// TIA Portal V20 export
FUNCTION "CollectAlarms" : Void   // FC85, LAD
TITLE = Alarm Collector Unit
// Collects alarms from the respective level and categorises the alarms into the different alarm classes.
// stored: Namespace Unit1.Em7, SetENOAutomatically false
   VAR_INPUT
      resetAlarms : Bool;
      disableAlarms : Bool;
   END_VAR
   VAR_OUTPUT
      commandsToUnit : "LUC_typeStateCommands";   // Feedback to the unit
   END_VAR
   VAR CONSTANT
      DelayTime : Time := T#100ms;
      NoDelayTime : Time;
      TRUE : Bool := TRUE;
      FALSE : Bool := FALSE;
   END_VAR
   VAR_TEMP   // added for the SCL form of the ladder/FBD networks
      _w1 : Bool;
   END_VAR
BEGIN

REGION Network 1: Reset Alarms
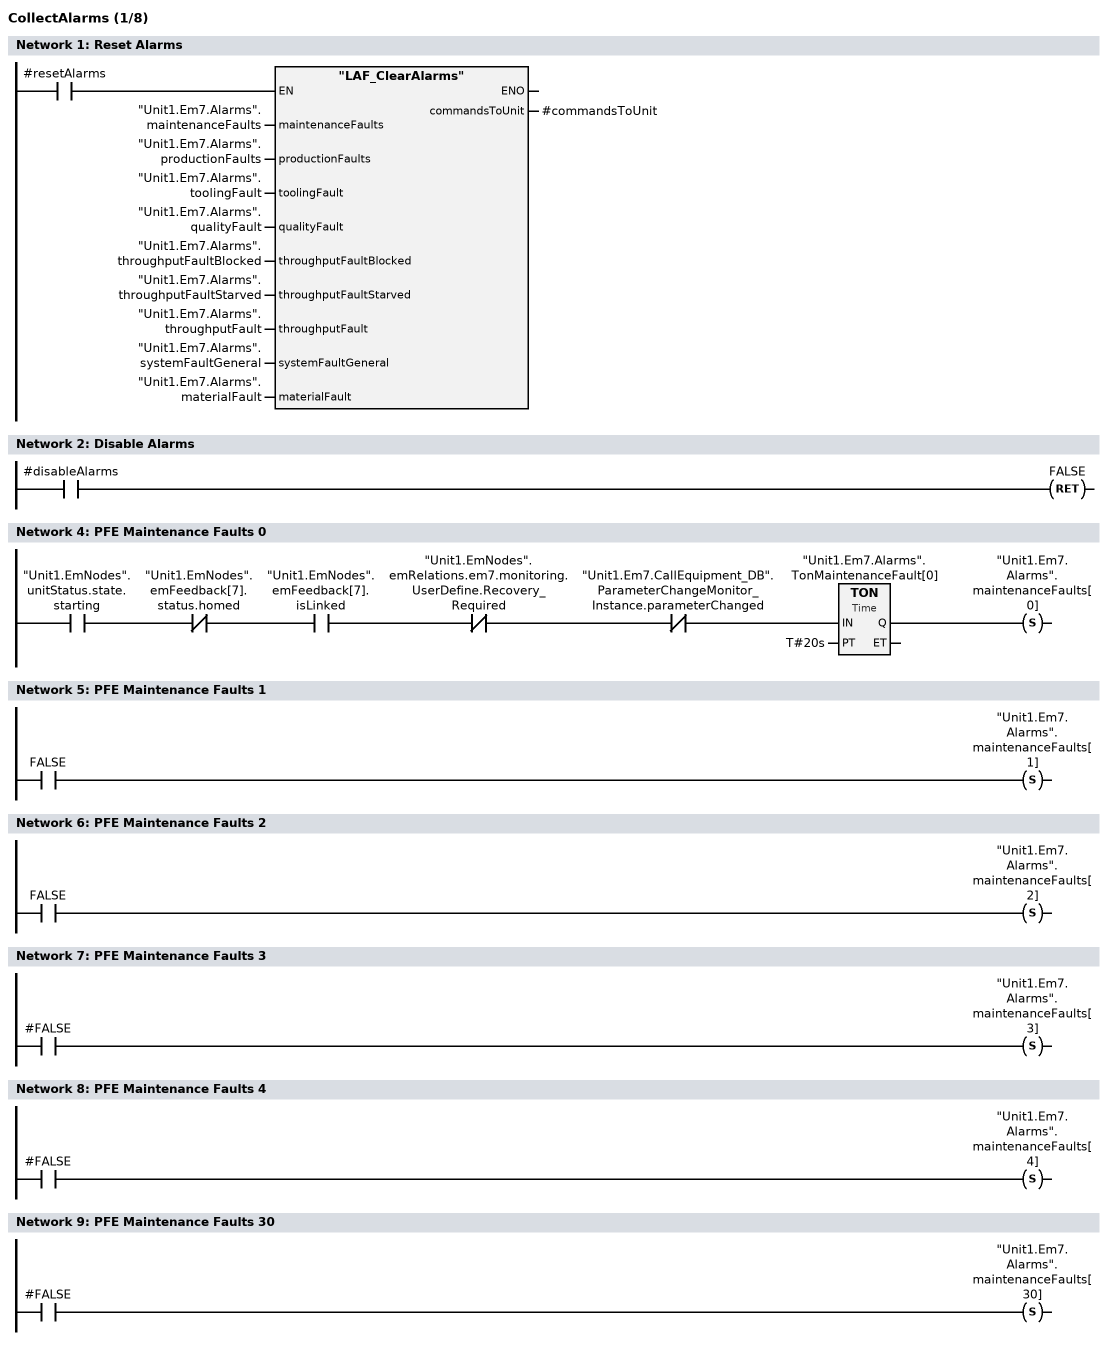
   RUNG wire#powerrail
      Contact( #resetAlarms )
      "LAF_ClearAlarms"(maintenanceFaults := "Unit1.Em7.Alarms".maintenanceFaults, productionFaults := "Unit1.Em7.Alarms".productionFaults, toolingFault := "Unit1.Em7.Alarms".toolingFault, qualityFault := "Unit1.Em7.Alarms".qualityFault, throughputFaultBlocked := "Unit1.Em7.Alarms".throughputFaultBlocked, throughputFaultStarved := "Unit1.Em7.Alarms".throughputFaultStarved, throughputFault := "Unit1.Em7.Alarms".throughputFault, systemFaultGeneral := "Unit1.Em7.Alarms".systemFaultGeneral, materialFault := "Unit1.Em7.Alarms".materialFault, commandsToUnit => #commandsToUnit)
   END_RUNG
   // the same network as SCL:
   IF #resetAlarms THEN
       "LAF_ClearAlarms"(maintenanceFaults := "Unit1.Em7.Alarms".maintenanceFaults,
                         productionFaults := "Unit1.Em7.Alarms".productionFaults,
                         toolingFault := "Unit1.Em7.Alarms".toolingFault,
                         qualityFault := "Unit1.Em7.Alarms".qualityFault,
                         throughputFaultBlocked := "Unit1.Em7.Alarms".throughputFaultBlocked,
                         throughputFaultStarved := "Unit1.Em7.Alarms".throughputFaultStarved,
                         throughputFault := "Unit1.Em7.Alarms".throughputFault,
                         systemFaultGeneral := "Unit1.Em7.Alarms".systemFaultGeneral,
                         materialFault := "Unit1.Em7.Alarms".materialFault,
                         commandsToUnit => #commandsToUnit);
   END_IF;
END_REGION

REGION Network 2: Disable Alarms
   RUNG wire#powerrail
      Contact( #disableAlarms )
      ReturnCoil( FALSE )
   END_RUNG
   // the same network as SCL:
   IF #disableAlarms THEN
       ENO := FALSE;
       RETURN;
   END_IF;
END_REGION

REGION Network 3: *************** Fault ************************
END_REGION

REGION Network 4: PFE Maintenance Faults 0
   RUNG wire#powerrail
      Contact( "Unit1.EmNodes".unitStatus.state.starting )
      I_Contact( "Unit1.EmNodes".emFeedback[7].status.homed )
      Contact( "Unit1.EmNodes".emFeedback[7].isLinked )
      I_Contact( "Unit1.EmNodes".emRelations.em7.monitoring.UserDefine.Recovery_Required )
      I_Contact( "Unit1.Em7.CallEquipment_DB".ParameterChangeMonitor_Instance.parameterChanged )
      { S7_Templates := "time_type := Time" } "Unit1.Em7.Alarms".TonMaintenanceFault[0].TON(pt := T#20s, et =>)
      S_Coil( "Unit1.Em7.Alarms".maintenanceFaults[0] )
   END_RUNG
   // the same network as SCL:
   "Unit1.Em7.Alarms".TonMaintenanceFault[0].TON(IN := "Unit1.EmNodes".unitStatus.state.starting AND NOT "Unit1.EmNodes".emFeedback[7].status.homed AND "Unit1.EmNodes".emFeedback[7].isLinked AND NOT "Unit1.EmNodes".emRelations.em7.monitoring.UserDefine.Recovery_Required AND NOT "Unit1.Em7.CallEquipment_DB".ParameterChangeMonitor_Instance.parameterChanged,
                           PT := T#20s);
   IF "Unit1.Em7.Alarms".TonMaintenanceFault[0].Q THEN
       "Unit1.Em7.Alarms".maintenanceFaults[0] := TRUE;
   END_IF;
END_REGION

REGION Network 5: PFE Maintenance Faults 1
   RUNG wire#powerrail
      Contact( FALSE )
      S_Coil( "Unit1.Em7.Alarms".maintenanceFaults[1] )
   END_RUNG
   // the same network as SCL:
   IF FALSE THEN "Unit1.Em7.Alarms".maintenanceFaults[1] := TRUE; END_IF;
END_REGION

REGION Network 6: PFE Maintenance Faults 2
   RUNG wire#powerrail
      Contact( FALSE )
      S_Coil( "Unit1.Em7.Alarms".maintenanceFaults[2] )
   END_RUNG
   // the same network as SCL:
   IF FALSE THEN "Unit1.Em7.Alarms".maintenanceFaults[2] := TRUE; END_IF;
END_REGION

REGION Network 7: PFE Maintenance Faults 3
   RUNG wire#powerrail
      Contact( #FALSE )
      S_Coil( "Unit1.Em7.Alarms".maintenanceFaults[3] )
   END_RUNG
   // the same network as SCL:
   IF #FALSE THEN "Unit1.Em7.Alarms".maintenanceFaults[3] := TRUE; END_IF;
END_REGION

REGION Network 8: PFE Maintenance Faults 4
   RUNG wire#powerrail
      Contact( #FALSE )
      S_Coil( "Unit1.Em7.Alarms".maintenanceFaults[4] )
   END_RUNG
   // the same network as SCL:
   IF #FALSE THEN "Unit1.Em7.Alarms".maintenanceFaults[4] := TRUE; END_IF;
END_REGION

REGION Network 9: PFE Maintenance Faults 30
   RUNG wire#powerrail
      Contact( #FALSE )
      S_Coil( "Unit1.Em7.Alarms".maintenanceFaults[30] )
   END_RUNG
   // the same network as SCL:
   IF #FALSE THEN "Unit1.Em7.Alarms".maintenanceFaults[30] := TRUE; END_IF;
END_REGION

REGION Network 10: PFE Maintenance Faults 31
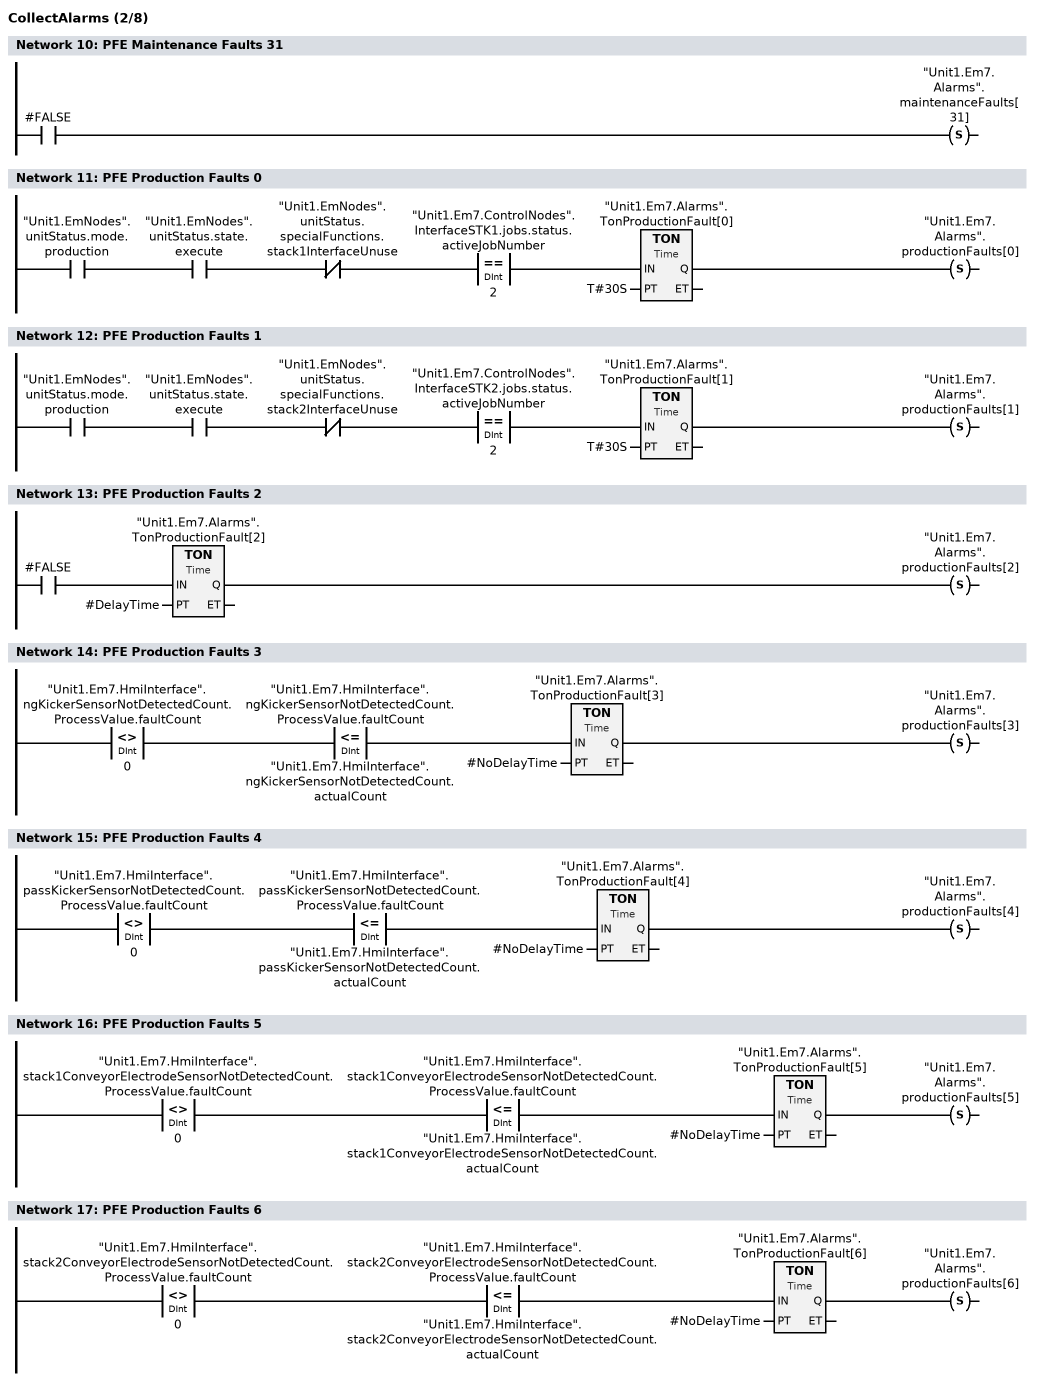
   RUNG wire#powerrail
      Contact( #FALSE )
      S_Coil( "Unit1.Em7.Alarms".maintenanceFaults[31] )
   END_RUNG
   // the same network as SCL:
   IF #FALSE THEN "Unit1.Em7.Alarms".maintenanceFaults[31] := TRUE; END_IF;
END_REGION

REGION Network 11: PFE Production Faults 0
   RUNG wire#powerrail
      Contact( "Unit1.EmNodes".unitStatus.mode.production )
      Contact( "Unit1.EmNodes".unitStatus.state.execute )
      I_Contact( "Unit1.EmNodes".unitStatus.specialFunctions.stack1InterfaceUnuse )
      { S7_Templates := "SrcType := DInt" } EQ_Contact(in1 := "Unit1.Em7.ControlNodes".InterfaceSTK1.jobs.status.activeJobNumber, in2 := 2)
      { S7_Templates := "time_type := Time" } "Unit1.Em7.Alarms".TonProductionFault[0].TON(pt := T#30S, et =>)
      S_Coil( "Unit1.Em7.Alarms".productionFaults[0] )
   END_RUNG
   // the same network as SCL:
   "Unit1.Em7.Alarms".TonProductionFault[0].TON(IN := "Unit1.EmNodes".unitStatus.mode.production AND "Unit1.EmNodes".unitStatus.state.execute AND NOT "Unit1.EmNodes".unitStatus.specialFunctions.stack1InterfaceUnuse AND ("Unit1.Em7.ControlNodes".InterfaceSTK1.jobs.status.activeJobNumber = 2),
                           PT := T#30S);
   IF "Unit1.Em7.Alarms".TonProductionFault[0].Q THEN "Unit1.Em7.Alarms".productionFaults[0] := TRUE; END_IF;
END_REGION

REGION Network 12: PFE Production Faults 1
   RUNG wire#powerrail
      Contact( "Unit1.EmNodes".unitStatus.mode.production )
      Contact( "Unit1.EmNodes".unitStatus.state.execute )
      I_Contact( "Unit1.EmNodes".unitStatus.specialFunctions.stack2InterfaceUnuse )
      { S7_Templates := "SrcType := DInt" } EQ_Contact(in1 := "Unit1.Em7.ControlNodes".InterfaceSTK2.jobs.status.activeJobNumber, in2 := 2)
      { S7_Templates := "time_type := Time" } "Unit1.Em7.Alarms".TonProductionFault[1].TON(pt := T#30S, et =>)
      S_Coil( "Unit1.Em7.Alarms".productionFaults[1] )
   END_RUNG
   // the same network as SCL:
   "Unit1.Em7.Alarms".TonProductionFault[1].TON(IN := "Unit1.EmNodes".unitStatus.mode.production AND "Unit1.EmNodes".unitStatus.state.execute AND NOT "Unit1.EmNodes".unitStatus.specialFunctions.stack2InterfaceUnuse AND ("Unit1.Em7.ControlNodes".InterfaceSTK2.jobs.status.activeJobNumber = 2),
                           PT := T#30S);
   IF "Unit1.Em7.Alarms".TonProductionFault[1].Q THEN "Unit1.Em7.Alarms".productionFaults[1] := TRUE; END_IF;
END_REGION

REGION Network 13: PFE Production Faults 2
   RUNG wire#powerrail
      Contact( #FALSE )
      { S7_Templates := "time_type := Time" } "Unit1.Em7.Alarms".TonProductionFault[2].TON(pt := #DelayTime, et =>)
      S_Coil( "Unit1.Em7.Alarms".productionFaults[2] )
   END_RUNG
   // the same network as SCL:
   "Unit1.Em7.Alarms".TonProductionFault[2].TON(IN := #FALSE, PT := #DelayTime);
   IF "Unit1.Em7.Alarms".TonProductionFault[2].Q THEN "Unit1.Em7.Alarms".productionFaults[2] := TRUE; END_IF;
END_REGION

REGION Network 14: PFE Production Faults 3
   RUNG wire#powerrail
      { S7_Templates := "SrcType := DInt" } NE_Contact(in1 := "Unit1.Em7.HmiInterface".ngKickerSensorNotDetectedCount.ProcessValue.faultCount, in2 := 0)
      { S7_Templates := "SrcType := DInt" } LE_Contact(in1 := "Unit1.Em7.HmiInterface".ngKickerSensorNotDetectedCount.ProcessValue.faultCount, in2 := "Unit1.Em7.HmiInterface".ngKickerSensorNotDetectedCount.actualCount)
      { S7_Templates := "time_type := Time" } "Unit1.Em7.Alarms".TonProductionFault[3].TON(pt := #NoDelayTime, et =>)
      S_Coil( "Unit1.Em7.Alarms".productionFaults[3] )
   END_RUNG
   // the same network as SCL:
   "Unit1.Em7.Alarms".TonProductionFault[3].TON(IN := ("Unit1.Em7.HmiInterface".ngKickerSensorNotDetectedCount.ProcessValue.faultCount <> 0) AND ("Unit1.Em7.HmiInterface".ngKickerSensorNotDetectedCount.ProcessValue.faultCount <= "Unit1.Em7.HmiInterface".ngKickerSensorNotDetectedCount.actualCount),
                           PT := #NoDelayTime);
   IF "Unit1.Em7.Alarms".TonProductionFault[3].Q THEN "Unit1.Em7.Alarms".productionFaults[3] := TRUE; END_IF;
END_REGION

REGION Network 15: PFE Production Faults 4
   RUNG wire#powerrail
      { S7_Templates := "SrcType := DInt" } NE_Contact(in1 := "Unit1.Em7.HmiInterface".passKickerSensorNotDetectedCount.ProcessValue.faultCount, in2 := 0)
      { S7_Templates := "SrcType := DInt" } LE_Contact(in1 := "Unit1.Em7.HmiInterface".passKickerSensorNotDetectedCount.ProcessValue.faultCount, in2 := "Unit1.Em7.HmiInterface".passKickerSensorNotDetectedCount.actualCount)
      { S7_Templates := "time_type := Time" } "Unit1.Em7.Alarms".TonProductionFault[4].TON(pt := #NoDelayTime, et =>)
      S_Coil( "Unit1.Em7.Alarms".productionFaults[4] )
   END_RUNG
   // the same network as SCL:
   "Unit1.Em7.Alarms".TonProductionFault[4].TON(IN := ("Unit1.Em7.HmiInterface".passKickerSensorNotDetectedCount.ProcessValue.faultCount <> 0) AND ("Unit1.Em7.HmiInterface".passKickerSensorNotDetectedCount.ProcessValue.faultCount <= "Unit1.Em7.HmiInterface".passKickerSensorNotDetectedCount.actualCount),
                           PT := #NoDelayTime);
   IF "Unit1.Em7.Alarms".TonProductionFault[4].Q THEN "Unit1.Em7.Alarms".productionFaults[4] := TRUE; END_IF;
END_REGION

REGION Network 16: PFE Production Faults 5
   RUNG wire#powerrail
      { S7_Templates := "SrcType := DInt" } NE_Contact(in1 := "Unit1.Em7.HmiInterface".stack1ConveyorElectrodeSensorNotDetectedCount.ProcessValue.faultCount, in2 := 0)
      { S7_Templates := "SrcType := DInt" } LE_Contact(in1 := "Unit1.Em7.HmiInterface".stack1ConveyorElectrodeSensorNotDetectedCount.ProcessValue.faultCount, in2 := "Unit1.Em7.HmiInterface".stack1ConveyorElectrodeSensorNotDetectedCount.actualCount)
      { S7_Templates := "time_type := Time" } "Unit1.Em7.Alarms".TonProductionFault[5].TON(pt := #NoDelayTime, et =>)
      S_Coil( "Unit1.Em7.Alarms".productionFaults[5] )
   END_RUNG
   // the same network as SCL:
   "Unit1.Em7.Alarms".TonProductionFault[5].TON(IN := ("Unit1.Em7.HmiInterface".stack1ConveyorElectrodeSensorNotDetectedCount.ProcessValue.faultCount <> 0) AND ("Unit1.Em7.HmiInterface".stack1ConveyorElectrodeSensorNotDetectedCount.ProcessValue.faultCount <= "Unit1.Em7.HmiInterface".stack1ConveyorElectrodeSensorNotDetectedCount.actualCount),
                           PT := #NoDelayTime);
   IF "Unit1.Em7.Alarms".TonProductionFault[5].Q THEN "Unit1.Em7.Alarms".productionFaults[5] := TRUE; END_IF;
END_REGION

REGION Network 17: PFE Production Faults 6
   RUNG wire#powerrail
      { S7_Templates := "SrcType := DInt" } NE_Contact(in1 := "Unit1.Em7.HmiInterface".stack2ConveyorElectrodeSensorNotDetectedCount.ProcessValue.faultCount, in2 := 0)
      { S7_Templates := "SrcType := DInt" } LE_Contact(in1 := "Unit1.Em7.HmiInterface".stack2ConveyorElectrodeSensorNotDetectedCount.ProcessValue.faultCount, in2 := "Unit1.Em7.HmiInterface".stack2ConveyorElectrodeSensorNotDetectedCount.actualCount)
      { S7_Templates := "time_type := Time" } "Unit1.Em7.Alarms".TonProductionFault[6].TON(pt := #NoDelayTime, et =>)
      S_Coil( "Unit1.Em7.Alarms".productionFaults[6] )
   END_RUNG
   // the same network as SCL:
   "Unit1.Em7.Alarms".TonProductionFault[6].TON(IN := ("Unit1.Em7.HmiInterface".stack2ConveyorElectrodeSensorNotDetectedCount.ProcessValue.faultCount <> 0) AND ("Unit1.Em7.HmiInterface".stack2ConveyorElectrodeSensorNotDetectedCount.ProcessValue.faultCount <= "Unit1.Em7.HmiInterface".stack2ConveyorElectrodeSensorNotDetectedCount.actualCount),
                           PT := #NoDelayTime);
   IF "Unit1.Em7.Alarms".TonProductionFault[6].Q THEN "Unit1.Em7.Alarms".productionFaults[6] := TRUE; END_IF;
END_REGION

REGION Network 18: PFE Production Faults 7
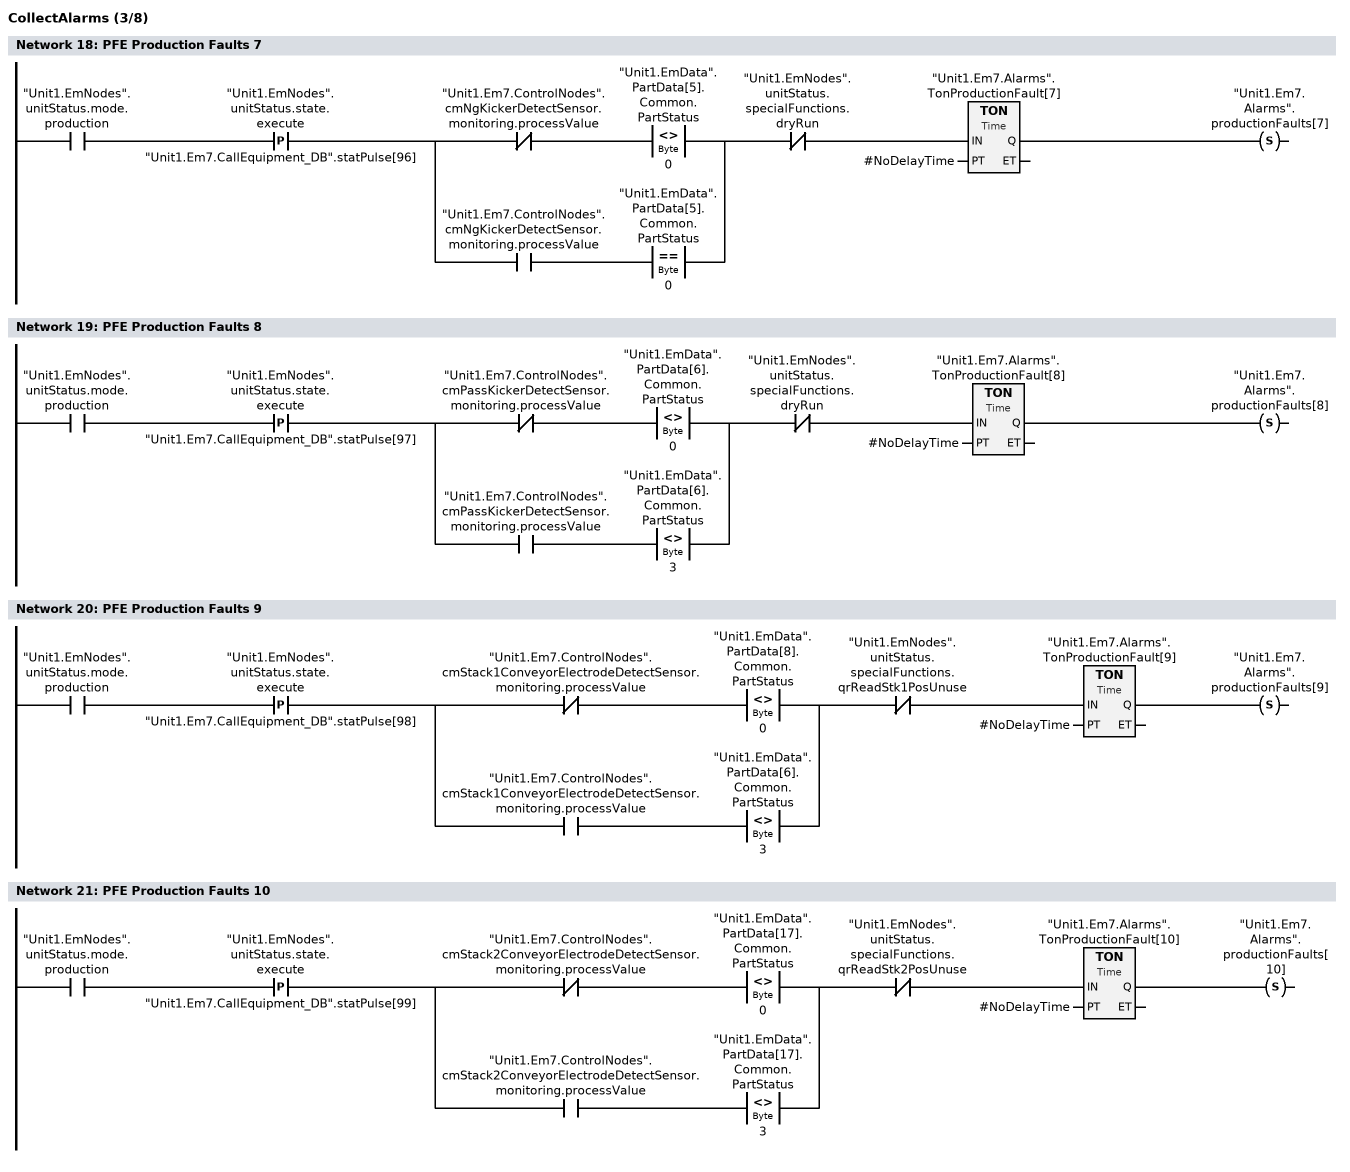
   RUNG wire#powerrail
      Contact( "Unit1.EmNodes".unitStatus.mode.production )
      P_Contact(operand := "Unit1.EmNodes".unitStatus.state.execute, bit := "Unit1.Em7.CallEquipment_DB".statPulse[96])
      wire#w1
      I_Contact( "Unit1.Em7.ControlNodes".cmNgKickerDetectSensor.monitoring.processValue )
      { S7_Templates := "SrcType := Byte" } NE_Contact(in1 := "Unit1.EmData".PartData[5].Common.PartStatus, in2 := 0)
      wire#w2
      I_Contact( "Unit1.EmNodes".unitStatus.specialFunctions.dryRun )
      { S7_Templates := "time_type := Time" } "Unit1.Em7.Alarms".TonProductionFault[7].TON(pt := #NoDelayTime, et =>)
      S_Coil( "Unit1.Em7.Alarms".productionFaults[7] )
   END_RUNG
   RUNG wire#w1
      Contact( "Unit1.Em7.ControlNodes".cmNgKickerDetectSensor.monitoring.processValue )
      { S7_Templates := "SrcType := Byte" } EQ_Contact(in1 := "Unit1.EmData".PartData[5].Common.PartStatus, in2 := 0)
   END_RUNG wire#w2
   // the same network as SCL:
   #_w1 := "Unit1.EmNodes".unitStatus.mode.production AND "Unit1.EmNodes".unitStatus.state.execute AND NOT "Unit1.Em7.CallEquipment_DB".statPulse[96];   // rising edge of "Unit1.EmNodes".unitStatus.state.execute
   "Unit1.Em7.CallEquipment_DB".statPulse[96] := "Unit1.EmNodes".unitStatus.state.execute;
   "Unit1.Em7.Alarms".TonProductionFault[7].TON(IN := #_w1 AND ((NOT "Unit1.Em7.ControlNodes".cmNgKickerDetectSensor.monitoring.processValue AND ("Unit1.EmData".PartData[5].Common.PartStatus <> 0)) OR ("Unit1.Em7.ControlNodes".cmNgKickerDetectSensor.monitoring.processValue AND ("Unit1.EmData".PartData[5].Common.PartStatus = 0))) AND NOT "Unit1.EmNodes".unitStatus.specialFunctions.dryRun,
                           PT := #NoDelayTime);
   IF "Unit1.Em7.Alarms".TonProductionFault[7].Q THEN "Unit1.Em7.Alarms".productionFaults[7] := TRUE; END_IF;
END_REGION

REGION Network 19: PFE Production Faults 8
   RUNG wire#powerrail
      Contact( "Unit1.EmNodes".unitStatus.mode.production )
      P_Contact(operand := "Unit1.EmNodes".unitStatus.state.execute, bit := "Unit1.Em7.CallEquipment_DB".statPulse[97])
      wire#w1
      I_Contact( "Unit1.Em7.ControlNodes".cmPassKickerDetectSensor.monitoring.processValue )
      { S7_Templates := "SrcType := Byte" } NE_Contact(in1 := "Unit1.EmData".PartData[6].Common.PartStatus, in2 := 0)
      wire#w2
      I_Contact( "Unit1.EmNodes".unitStatus.specialFunctions.dryRun )
      { S7_Templates := "time_type := Time" } "Unit1.Em7.Alarms".TonProductionFault[8].TON(pt := #NoDelayTime, et =>)
      S_Coil( "Unit1.Em7.Alarms".productionFaults[8] )
   END_RUNG
   RUNG wire#w1
      Contact( "Unit1.Em7.ControlNodes".cmPassKickerDetectSensor.monitoring.processValue )
      { S7_Templates := "SrcType := Byte" } NE_Contact(in1 := "Unit1.EmData".PartData[6].Common.PartStatus, in2 := 3)
   END_RUNG wire#w2
   // the same network as SCL:
   #_w1 := "Unit1.EmNodes".unitStatus.mode.production AND "Unit1.EmNodes".unitStatus.state.execute AND NOT "Unit1.Em7.CallEquipment_DB".statPulse[97];   // rising edge of "Unit1.EmNodes".unitStatus.state.execute
   "Unit1.Em7.CallEquipment_DB".statPulse[97] := "Unit1.EmNodes".unitStatus.state.execute;
   "Unit1.Em7.Alarms".TonProductionFault[8].TON(IN := #_w1 AND ((NOT "Unit1.Em7.ControlNodes".cmPassKickerDetectSensor.monitoring.processValue AND ("Unit1.EmData".PartData[6].Common.PartStatus <> 0)) OR ("Unit1.Em7.ControlNodes".cmPassKickerDetectSensor.monitoring.processValue AND ("Unit1.EmData".PartData[6].Common.PartStatus <> 3))) AND NOT "Unit1.EmNodes".unitStatus.specialFunctions.dryRun,
                           PT := #NoDelayTime);
   IF "Unit1.Em7.Alarms".TonProductionFault[8].Q THEN "Unit1.Em7.Alarms".productionFaults[8] := TRUE; END_IF;
END_REGION

REGION Network 20: PFE Production Faults 9
   RUNG wire#powerrail
      Contact( "Unit1.EmNodes".unitStatus.mode.production )
      P_Contact(operand := "Unit1.EmNodes".unitStatus.state.execute, bit := "Unit1.Em7.CallEquipment_DB".statPulse[98])
      wire#w1
      I_Contact( "Unit1.Em7.ControlNodes".cmStack1ConveyorElectrodeDetectSensor.monitoring.processValue )
      { S7_Templates := "SrcType := Byte" } NE_Contact(in1 := "Unit1.EmData".PartData[8].Common.PartStatus, in2 := 0)
      wire#w2
      I_Contact( "Unit1.EmNodes".unitStatus.specialFunctions.qrReadStk1PosUnuse )
      { S7_Templates := "time_type := Time" } "Unit1.Em7.Alarms".TonProductionFault[9].TON(pt := #NoDelayTime, et =>)
      S_Coil( "Unit1.Em7.Alarms".productionFaults[9] )
   END_RUNG
   RUNG wire#w1
      Contact( "Unit1.Em7.ControlNodes".cmStack1ConveyorElectrodeDetectSensor.monitoring.processValue )
      { S7_Templates := "SrcType := Byte" } NE_Contact(in1 := "Unit1.EmData".PartData[6].Common.PartStatus, in2 := 3)
   END_RUNG wire#w2
   // the same network as SCL:
   #_w1 := "Unit1.EmNodes".unitStatus.mode.production AND "Unit1.EmNodes".unitStatus.state.execute AND NOT "Unit1.Em7.CallEquipment_DB".statPulse[98];   // rising edge of "Unit1.EmNodes".unitStatus.state.execute
   "Unit1.Em7.CallEquipment_DB".statPulse[98] := "Unit1.EmNodes".unitStatus.state.execute;
   "Unit1.Em7.Alarms".TonProductionFault[9].TON(IN := #_w1 AND ((NOT "Unit1.Em7.ControlNodes".cmStack1ConveyorElectrodeDetectSensor.monitoring.processValue AND ("Unit1.EmData".PartData[8].Common.PartStatus <> 0)) OR ("Unit1.Em7.ControlNodes".cmStack1ConveyorElectrodeDetectSensor.monitoring.processValue AND ("Unit1.EmData".PartData[6].Common.PartStatus <> 3))) AND NOT "Unit1.EmNodes".unitStatus.specialFunctions.qrReadStk1PosUnuse,
                           PT := #NoDelayTime);
   IF "Unit1.Em7.Alarms".TonProductionFault[9].Q THEN "Unit1.Em7.Alarms".productionFaults[9] := TRUE; END_IF;
END_REGION

REGION Network 21: PFE Production Faults 10
   RUNG wire#powerrail
      Contact( "Unit1.EmNodes".unitStatus.mode.production )
      P_Contact(operand := "Unit1.EmNodes".unitStatus.state.execute, bit := "Unit1.Em7.CallEquipment_DB".statPulse[99])
      wire#w1
      I_Contact( "Unit1.Em7.ControlNodes".cmStack2ConveyorElectrodeDetectSensor.monitoring.processValue )
      { S7_Templates := "SrcType := Byte" } NE_Contact(in1 := "Unit1.EmData".PartData[17].Common.PartStatus, in2 := 0)
      wire#w2
      I_Contact( "Unit1.EmNodes".unitStatus.specialFunctions.qrReadStk2PosUnuse )
      { S7_Templates := "time_type := Time" } "Unit1.Em7.Alarms".TonProductionFault[10].TON(pt := #NoDelayTime, et =>)
      S_Coil( "Unit1.Em7.Alarms".productionFaults[10] )
   END_RUNG
   RUNG wire#w1
      Contact( "Unit1.Em7.ControlNodes".cmStack2ConveyorElectrodeDetectSensor.monitoring.processValue )
      { S7_Templates := "SrcType := Byte" } NE_Contact(in1 := "Unit1.EmData".PartData[17].Common.PartStatus, in2 := 3)
   END_RUNG wire#w2
   // the same network as SCL:
   #_w1 := "Unit1.EmNodes".unitStatus.mode.production AND "Unit1.EmNodes".unitStatus.state.execute AND NOT "Unit1.Em7.CallEquipment_DB".statPulse[99];   // rising edge of "Unit1.EmNodes".unitStatus.state.execute
   "Unit1.Em7.CallEquipment_DB".statPulse[99] := "Unit1.EmNodes".unitStatus.state.execute;
   "Unit1.Em7.Alarms".TonProductionFault[10].TON(IN := #_w1 AND ((NOT "Unit1.Em7.ControlNodes".cmStack2ConveyorElectrodeDetectSensor.monitoring.processValue AND ("Unit1.EmData".PartData[17].Common.PartStatus <> 0)) OR ("Unit1.Em7.ControlNodes".cmStack2ConveyorElectrodeDetectSensor.monitoring.processValue AND ("Unit1.EmData".PartData[17].Common.PartStatus <> 3))) AND NOT "Unit1.EmNodes".unitStatus.specialFunctions.qrReadStk2PosUnuse,
                           PT := #NoDelayTime);
   IF "Unit1.Em7.Alarms".TonProductionFault[10].Q THEN
       "Unit1.Em7.Alarms".productionFaults[10] := TRUE;
   END_IF;
END_REGION

REGION Network 22: PFE Production Faults 11
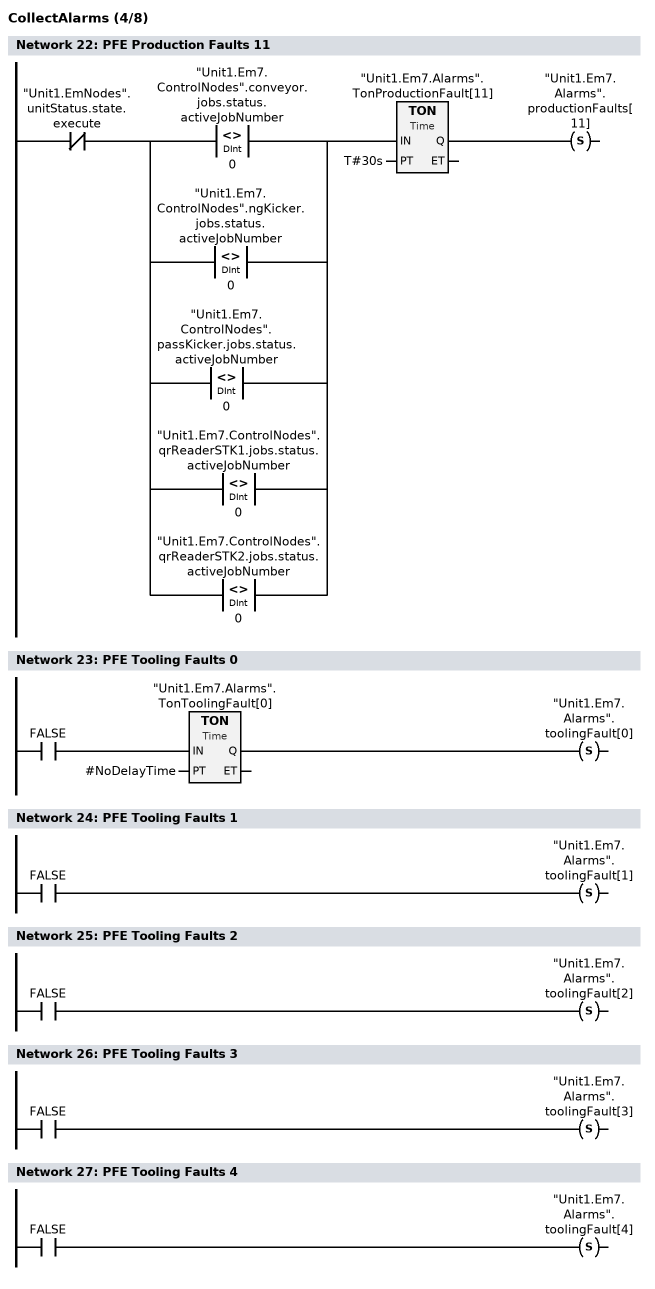
   RUNG wire#powerrail
      I_Contact( "Unit1.EmNodes".unitStatus.state.execute )
      wire#w1
      { S7_Templates := "SrcType := DInt" } NE_Contact(in1 := "Unit1.Em7.ControlNodes".conveyor.jobs.status.activeJobNumber, in2 := 0)
      wire#w2
      { S7_Templates := "time_type := Time" } "Unit1.Em7.Alarms".TonProductionFault[11].TON(pt := T#30s, et =>)
      S_Coil( "Unit1.Em7.Alarms".productionFaults[11] )
   END_RUNG
   RUNG wire#w1
      { S7_Templates := "SrcType := DInt" } NE_Contact(in1 := "Unit1.Em7.ControlNodes".ngKicker.jobs.status.activeJobNumber, in2 := 0)
   END_RUNG wire#w2
   RUNG wire#w1
      { S7_Templates := "SrcType := DInt" } NE_Contact(in1 := "Unit1.Em7.ControlNodes".passKicker.jobs.status.activeJobNumber, in2 := 0)
   END_RUNG wire#w2
   RUNG wire#w1
      { S7_Templates := "SrcType := DInt" } NE_Contact(in1 := "Unit1.Em7.ControlNodes".qrReaderSTK1.jobs.status.activeJobNumber, in2 := 0)
   END_RUNG wire#w2
   RUNG wire#w1
      { S7_Templates := "SrcType := DInt" } NE_Contact(in1 := "Unit1.Em7.ControlNodes".qrReaderSTK2.jobs.status.activeJobNumber, in2 := 0)
   END_RUNG wire#w2
   // the same network as SCL:
   "Unit1.Em7.Alarms".TonProductionFault[11].TON(IN := NOT "Unit1.EmNodes".unitStatus.state.execute AND (("Unit1.Em7.ControlNodes".conveyor.jobs.status.activeJobNumber <> 0) OR ("Unit1.Em7.ControlNodes".ngKicker.jobs.status.activeJobNumber <> 0) OR ("Unit1.Em7.ControlNodes".passKicker.jobs.status.activeJobNumber <> 0) OR ("Unit1.Em7.ControlNodes".qrReaderSTK1.jobs.status.activeJobNumber <> 0) OR ("Unit1.Em7.ControlNodes".qrReaderSTK2.jobs.status.activeJobNumber <> 0)),
                           PT := T#30s);
   IF "Unit1.Em7.Alarms".TonProductionFault[11].Q THEN
       "Unit1.Em7.Alarms".productionFaults[11] := TRUE;
   END_IF;
END_REGION

REGION Network 23: PFE Tooling Faults 0
   RUNG wire#powerrail
      Contact( FALSE )
      { S7_Templates := "time_type := Time" } "Unit1.Em7.Alarms".TonToolingFault[0].TON(pt := #NoDelayTime, et =>)
      S_Coil( "Unit1.Em7.Alarms".toolingFault[0] )
   END_RUNG
   // the same network as SCL:
   "Unit1.Em7.Alarms".TonToolingFault[0].TON(IN := FALSE, PT := #NoDelayTime);
   IF "Unit1.Em7.Alarms".TonToolingFault[0].Q THEN "Unit1.Em7.Alarms".toolingFault[0] := TRUE; END_IF;
END_REGION

REGION Network 24: PFE Tooling Faults 1
   RUNG wire#powerrail
      Contact( FALSE )
      S_Coil( "Unit1.Em7.Alarms".toolingFault[1] )
   END_RUNG
   // the same network as SCL:
   IF FALSE THEN "Unit1.Em7.Alarms".toolingFault[1] := TRUE; END_IF;
END_REGION

REGION Network 25: PFE Tooling Faults 2
   RUNG wire#powerrail
      Contact( FALSE )
      S_Coil( "Unit1.Em7.Alarms".toolingFault[2] )
   END_RUNG
   // the same network as SCL:
   IF FALSE THEN "Unit1.Em7.Alarms".toolingFault[2] := TRUE; END_IF;
END_REGION

REGION Network 26: PFE Tooling Faults 3
   RUNG wire#powerrail
      Contact( FALSE )
      S_Coil( "Unit1.Em7.Alarms".toolingFault[3] )
   END_RUNG
   // the same network as SCL:
   IF FALSE THEN "Unit1.Em7.Alarms".toolingFault[3] := TRUE; END_IF;
END_REGION

REGION Network 27: PFE Tooling Faults 4
   RUNG wire#powerrail
      Contact( FALSE )
      S_Coil( "Unit1.Em7.Alarms".toolingFault[4] )
   END_RUNG
   // the same network as SCL:
   IF FALSE THEN "Unit1.Em7.Alarms".toolingFault[4] := TRUE; END_IF;
END_REGION

REGION Network 28: PFE Quality Faults 0
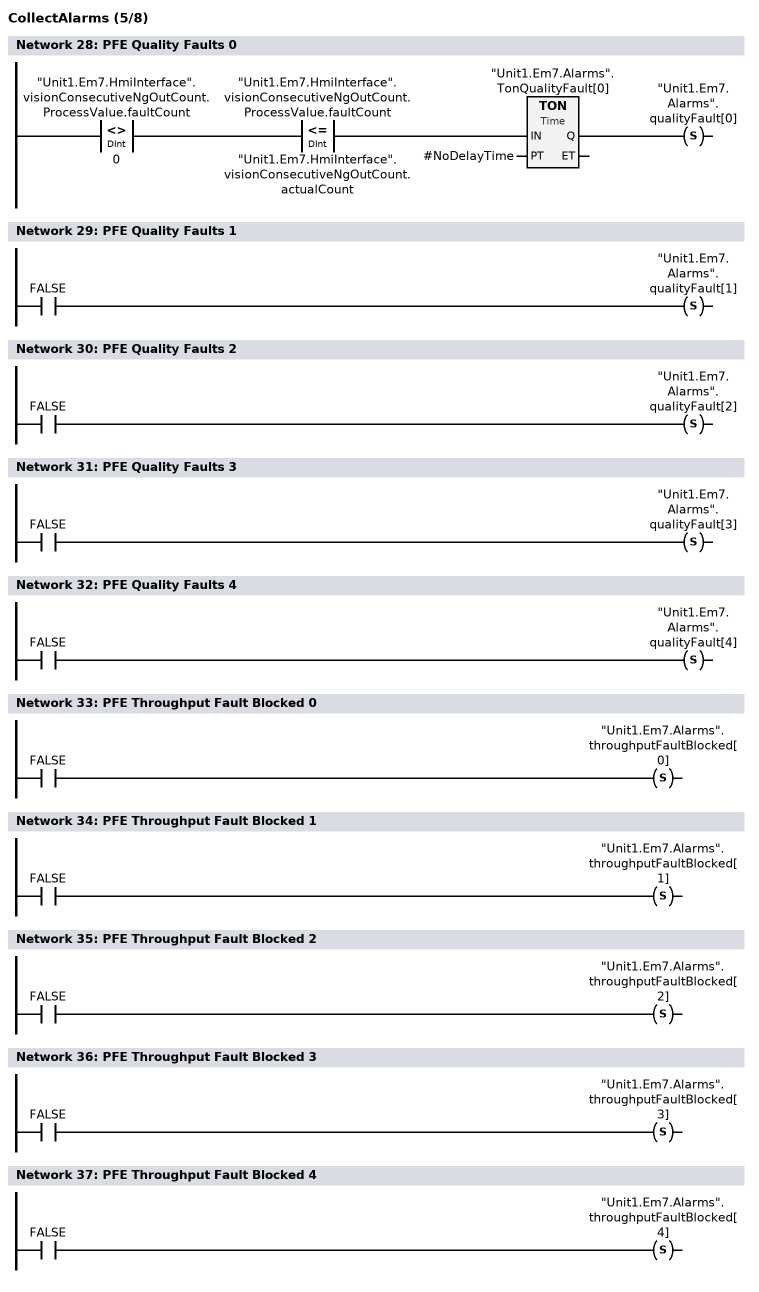
   RUNG wire#powerrail
      { S7_Templates := "SrcType := DInt" } NE_Contact(in1 := "Unit1.Em7.HmiInterface".visionConsecutiveNgOutCount.ProcessValue.faultCount, in2 := 0)
      { S7_Templates := "SrcType := DInt" } LE_Contact(in1 := "Unit1.Em7.HmiInterface".visionConsecutiveNgOutCount.ProcessValue.faultCount, in2 := "Unit1.Em7.HmiInterface".visionConsecutiveNgOutCount.actualCount)
      { S7_Templates := "time_type := Time" } "Unit1.Em7.Alarms".TonQualityFault[0].TON(pt := #NoDelayTime, et =>)
      S_Coil( "Unit1.Em7.Alarms".qualityFault[0] )
   END_RUNG
   // the same network as SCL:
   "Unit1.Em7.Alarms".TonQualityFault[0].TON(IN := ("Unit1.Em7.HmiInterface".visionConsecutiveNgOutCount.ProcessValue.faultCount <> 0) AND ("Unit1.Em7.HmiInterface".visionConsecutiveNgOutCount.ProcessValue.faultCount <= "Unit1.Em7.HmiInterface".visionConsecutiveNgOutCount.actualCount),
                           PT := #NoDelayTime);
   IF "Unit1.Em7.Alarms".TonQualityFault[0].Q THEN "Unit1.Em7.Alarms".qualityFault[0] := TRUE; END_IF;
END_REGION

REGION Network 29: PFE Quality Faults 1
   RUNG wire#powerrail
      Contact( FALSE )
      S_Coil( "Unit1.Em7.Alarms".qualityFault[1] )
   END_RUNG
   // the same network as SCL:
   IF FALSE THEN "Unit1.Em7.Alarms".qualityFault[1] := TRUE; END_IF;
END_REGION

REGION Network 30: PFE Quality Faults 2
   RUNG wire#powerrail
      Contact( FALSE )
      S_Coil( "Unit1.Em7.Alarms".qualityFault[2] )
   END_RUNG
   // the same network as SCL:
   IF FALSE THEN "Unit1.Em7.Alarms".qualityFault[2] := TRUE; END_IF;
END_REGION

REGION Network 31: PFE Quality Faults 3
   RUNG wire#powerrail
      Contact( FALSE )
      S_Coil( "Unit1.Em7.Alarms".qualityFault[3] )
   END_RUNG
   // the same network as SCL:
   IF FALSE THEN "Unit1.Em7.Alarms".qualityFault[3] := TRUE; END_IF;
END_REGION

REGION Network 32: PFE Quality Faults 4
   RUNG wire#powerrail
      Contact( FALSE )
      S_Coil( "Unit1.Em7.Alarms".qualityFault[4] )
   END_RUNG
   // the same network as SCL:
   IF FALSE THEN "Unit1.Em7.Alarms".qualityFault[4] := TRUE; END_IF;
END_REGION

REGION Network 33: PFE Throughput Fault Blocked 0
   RUNG wire#powerrail
      Contact( FALSE )
      S_Coil( "Unit1.Em7.Alarms".throughputFaultBlocked[0] )
   END_RUNG
   // the same network as SCL:
   IF FALSE THEN "Unit1.Em7.Alarms".throughputFaultBlocked[0] := TRUE; END_IF;
END_REGION

REGION Network 34: PFE Throughput Fault Blocked 1
   RUNG wire#powerrail
      Contact( FALSE )
      S_Coil( "Unit1.Em7.Alarms".throughputFaultBlocked[1] )
   END_RUNG
   // the same network as SCL:
   IF FALSE THEN "Unit1.Em7.Alarms".throughputFaultBlocked[1] := TRUE; END_IF;
END_REGION

REGION Network 35: PFE Throughput Fault Blocked 2
   RUNG wire#powerrail
      Contact( FALSE )
      S_Coil( "Unit1.Em7.Alarms".throughputFaultBlocked[2] )
   END_RUNG
   // the same network as SCL:
   IF FALSE THEN "Unit1.Em7.Alarms".throughputFaultBlocked[2] := TRUE; END_IF;
END_REGION

REGION Network 36: PFE Throughput Fault Blocked 3
   RUNG wire#powerrail
      Contact( FALSE )
      S_Coil( "Unit1.Em7.Alarms".throughputFaultBlocked[3] )
   END_RUNG
   // the same network as SCL:
   IF FALSE THEN "Unit1.Em7.Alarms".throughputFaultBlocked[3] := TRUE; END_IF;
END_REGION

REGION Network 37: PFE Throughput Fault Blocked 4
   RUNG wire#powerrail
      Contact( FALSE )
      S_Coil( "Unit1.Em7.Alarms".throughputFaultBlocked[4] )
   END_RUNG
   // the same network as SCL:
   IF FALSE THEN "Unit1.Em7.Alarms".throughputFaultBlocked[4] := TRUE; END_IF;
END_REGION

REGION Network 38: PFE Throughput Fault Starved 0
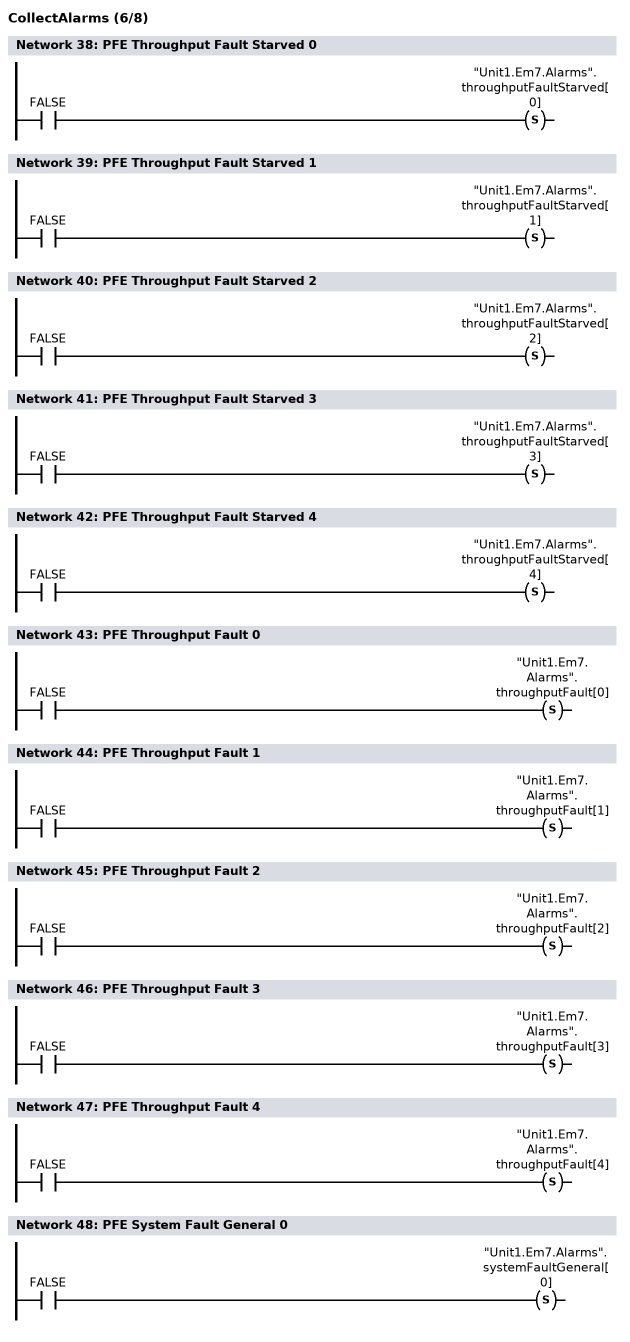
   RUNG wire#powerrail
      Contact( FALSE )
      S_Coil( "Unit1.Em7.Alarms".throughputFaultStarved[0] )
   END_RUNG
   // the same network as SCL:
   IF FALSE THEN "Unit1.Em7.Alarms".throughputFaultStarved[0] := TRUE; END_IF;
END_REGION

REGION Network 39: PFE Throughput Fault Starved 1
   RUNG wire#powerrail
      Contact( FALSE )
      S_Coil( "Unit1.Em7.Alarms".throughputFaultStarved[1] )
   END_RUNG
   // the same network as SCL:
   IF FALSE THEN "Unit1.Em7.Alarms".throughputFaultStarved[1] := TRUE; END_IF;
END_REGION

REGION Network 40: PFE Throughput Fault Starved 2
   RUNG wire#powerrail
      Contact( FALSE )
      S_Coil( "Unit1.Em7.Alarms".throughputFaultStarved[2] )
   END_RUNG
   // the same network as SCL:
   IF FALSE THEN "Unit1.Em7.Alarms".throughputFaultStarved[2] := TRUE; END_IF;
END_REGION

REGION Network 41: PFE Throughput Fault Starved 3
   RUNG wire#powerrail
      Contact( FALSE )
      S_Coil( "Unit1.Em7.Alarms".throughputFaultStarved[3] )
   END_RUNG
   // the same network as SCL:
   IF FALSE THEN "Unit1.Em7.Alarms".throughputFaultStarved[3] := TRUE; END_IF;
END_REGION

REGION Network 42: PFE Throughput Fault Starved 4
   RUNG wire#powerrail
      Contact( FALSE )
      S_Coil( "Unit1.Em7.Alarms".throughputFaultStarved[4] )
   END_RUNG
   // the same network as SCL:
   IF FALSE THEN "Unit1.Em7.Alarms".throughputFaultStarved[4] := TRUE; END_IF;
END_REGION

REGION Network 43: PFE Throughput Fault 0
   RUNG wire#powerrail
      Contact( FALSE )
      S_Coil( "Unit1.Em7.Alarms".throughputFault[0] )
   END_RUNG
   // the same network as SCL:
   IF FALSE THEN "Unit1.Em7.Alarms".throughputFault[0] := TRUE; END_IF;
END_REGION

REGION Network 44: PFE Throughput Fault 1
   RUNG wire#powerrail
      Contact( FALSE )
      S_Coil( "Unit1.Em7.Alarms".throughputFault[1] )
   END_RUNG
   // the same network as SCL:
   IF FALSE THEN "Unit1.Em7.Alarms".throughputFault[1] := TRUE; END_IF;
END_REGION

REGION Network 45: PFE Throughput Fault 2
   RUNG wire#powerrail
      Contact( FALSE )
      S_Coil( "Unit1.Em7.Alarms".throughputFault[2] )
   END_RUNG
   // the same network as SCL:
   IF FALSE THEN "Unit1.Em7.Alarms".throughputFault[2] := TRUE; END_IF;
END_REGION

REGION Network 46: PFE Throughput Fault 3
   RUNG wire#powerrail
      Contact( FALSE )
      S_Coil( "Unit1.Em7.Alarms".throughputFault[3] )
   END_RUNG
   // the same network as SCL:
   IF FALSE THEN "Unit1.Em7.Alarms".throughputFault[3] := TRUE; END_IF;
END_REGION

REGION Network 47: PFE Throughput Fault 4
   RUNG wire#powerrail
      Contact( FALSE )
      S_Coil( "Unit1.Em7.Alarms".throughputFault[4] )
   END_RUNG
   // the same network as SCL:
   IF FALSE THEN "Unit1.Em7.Alarms".throughputFault[4] := TRUE; END_IF;
END_REGION

REGION Network 48: PFE System Fault General 0
   RUNG wire#powerrail
      Contact( FALSE )
      S_Coil( "Unit1.Em7.Alarms".systemFaultGeneral[0] )
   END_RUNG
   // the same network as SCL:
   IF FALSE THEN "Unit1.Em7.Alarms".systemFaultGeneral[0] := TRUE; END_IF;
END_REGION

REGION Network 49: PFE System Fault General 1
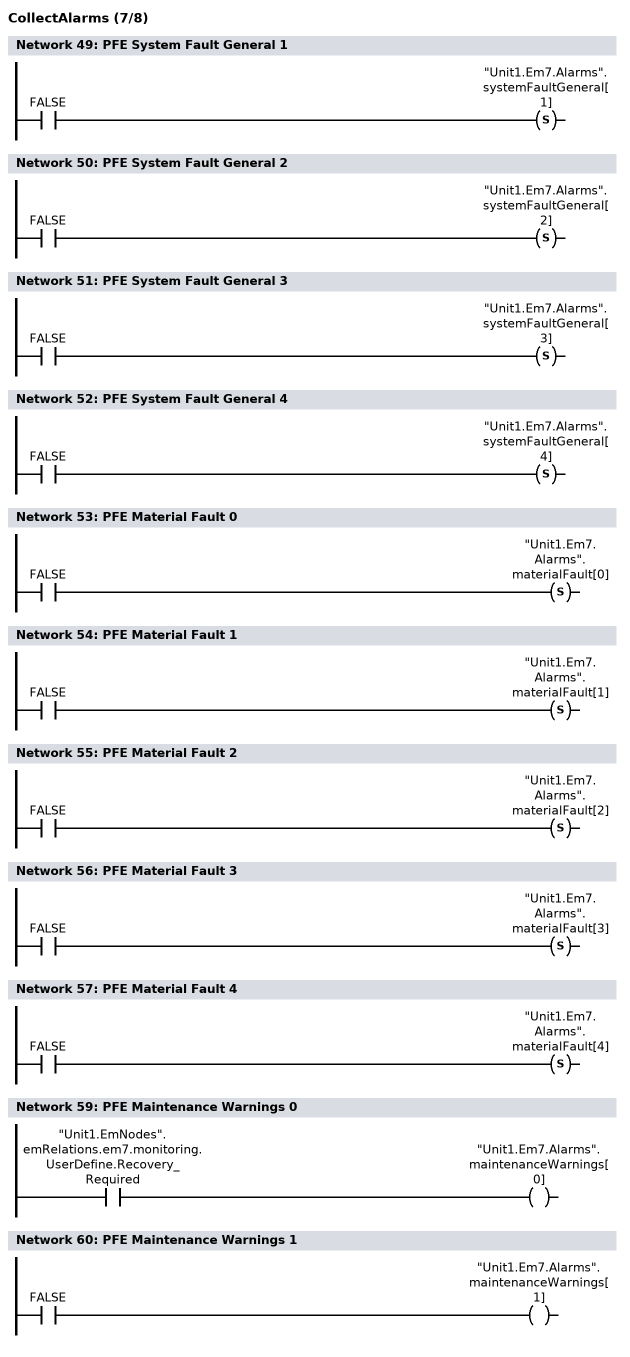
   RUNG wire#powerrail
      Contact( FALSE )
      S_Coil( "Unit1.Em7.Alarms".systemFaultGeneral[1] )
   END_RUNG
   // the same network as SCL:
   IF FALSE THEN "Unit1.Em7.Alarms".systemFaultGeneral[1] := TRUE; END_IF;
END_REGION

REGION Network 50: PFE System Fault General 2
   RUNG wire#powerrail
      Contact( FALSE )
      S_Coil( "Unit1.Em7.Alarms".systemFaultGeneral[2] )
   END_RUNG
   // the same network as SCL:
   IF FALSE THEN "Unit1.Em7.Alarms".systemFaultGeneral[2] := TRUE; END_IF;
END_REGION

REGION Network 51: PFE System Fault General 3
   RUNG wire#powerrail
      Contact( FALSE )
      S_Coil( "Unit1.Em7.Alarms".systemFaultGeneral[3] )
   END_RUNG
   // the same network as SCL:
   IF FALSE THEN "Unit1.Em7.Alarms".systemFaultGeneral[3] := TRUE; END_IF;
END_REGION

REGION Network 52: PFE System Fault General 4
   RUNG wire#powerrail
      Contact( FALSE )
      S_Coil( "Unit1.Em7.Alarms".systemFaultGeneral[4] )
   END_RUNG
   // the same network as SCL:
   IF FALSE THEN "Unit1.Em7.Alarms".systemFaultGeneral[4] := TRUE; END_IF;
END_REGION

REGION Network 53: PFE Material Fault 0
   RUNG wire#powerrail
      Contact( FALSE )
      S_Coil( "Unit1.Em7.Alarms".materialFault[0] )
   END_RUNG
   // the same network as SCL:
   IF FALSE THEN "Unit1.Em7.Alarms".materialFault[0] := TRUE; END_IF;
END_REGION

REGION Network 54: PFE Material Fault 1
   RUNG wire#powerrail
      Contact( FALSE )
      S_Coil( "Unit1.Em7.Alarms".materialFault[1] )
   END_RUNG
   // the same network as SCL:
   IF FALSE THEN "Unit1.Em7.Alarms".materialFault[1] := TRUE; END_IF;
END_REGION

REGION Network 55: PFE Material Fault 2
   RUNG wire#powerrail
      Contact( FALSE )
      S_Coil( "Unit1.Em7.Alarms".materialFault[2] )
   END_RUNG
   // the same network as SCL:
   IF FALSE THEN "Unit1.Em7.Alarms".materialFault[2] := TRUE; END_IF;
END_REGION

REGION Network 56: PFE Material Fault 3
   RUNG wire#powerrail
      Contact( FALSE )
      S_Coil( "Unit1.Em7.Alarms".materialFault[3] )
   END_RUNG
   // the same network as SCL:
   IF FALSE THEN "Unit1.Em7.Alarms".materialFault[3] := TRUE; END_IF;
END_REGION

REGION Network 57: PFE Material Fault 4
   RUNG wire#powerrail
      Contact( FALSE )
      S_Coil( "Unit1.Em7.Alarms".materialFault[4] )
   END_RUNG
   // the same network as SCL:
   IF FALSE THEN "Unit1.Em7.Alarms".materialFault[4] := TRUE; END_IF;
END_REGION

REGION Network 58: *************** Warning **************************
END_REGION

REGION Network 59: PFE Maintenance Warnings 0
   RUNG wire#powerrail
      Contact( "Unit1.EmNodes".emRelations.em7.monitoring.UserDefine.Recovery_Required )
      Coil( "Unit1.Em7.Alarms".maintenanceWarnings[0] )
   END_RUNG
   // the same network as SCL:
   "Unit1.Em7.Alarms".maintenanceWarnings[0] := "Unit1.EmNodes".emRelations.em7.monitoring.UserDefine.Recovery_Required;
END_REGION

REGION Network 60: PFE Maintenance Warnings 1
   RUNG wire#powerrail
      Contact( FALSE )
      Coil( "Unit1.Em7.Alarms".maintenanceWarnings[1] )
   END_RUNG
   // the same network as SCL:
   "Unit1.Em7.Alarms".maintenanceWarnings[1] := FALSE;
END_REGION

REGION Network 61: PFE Production Warnings 3
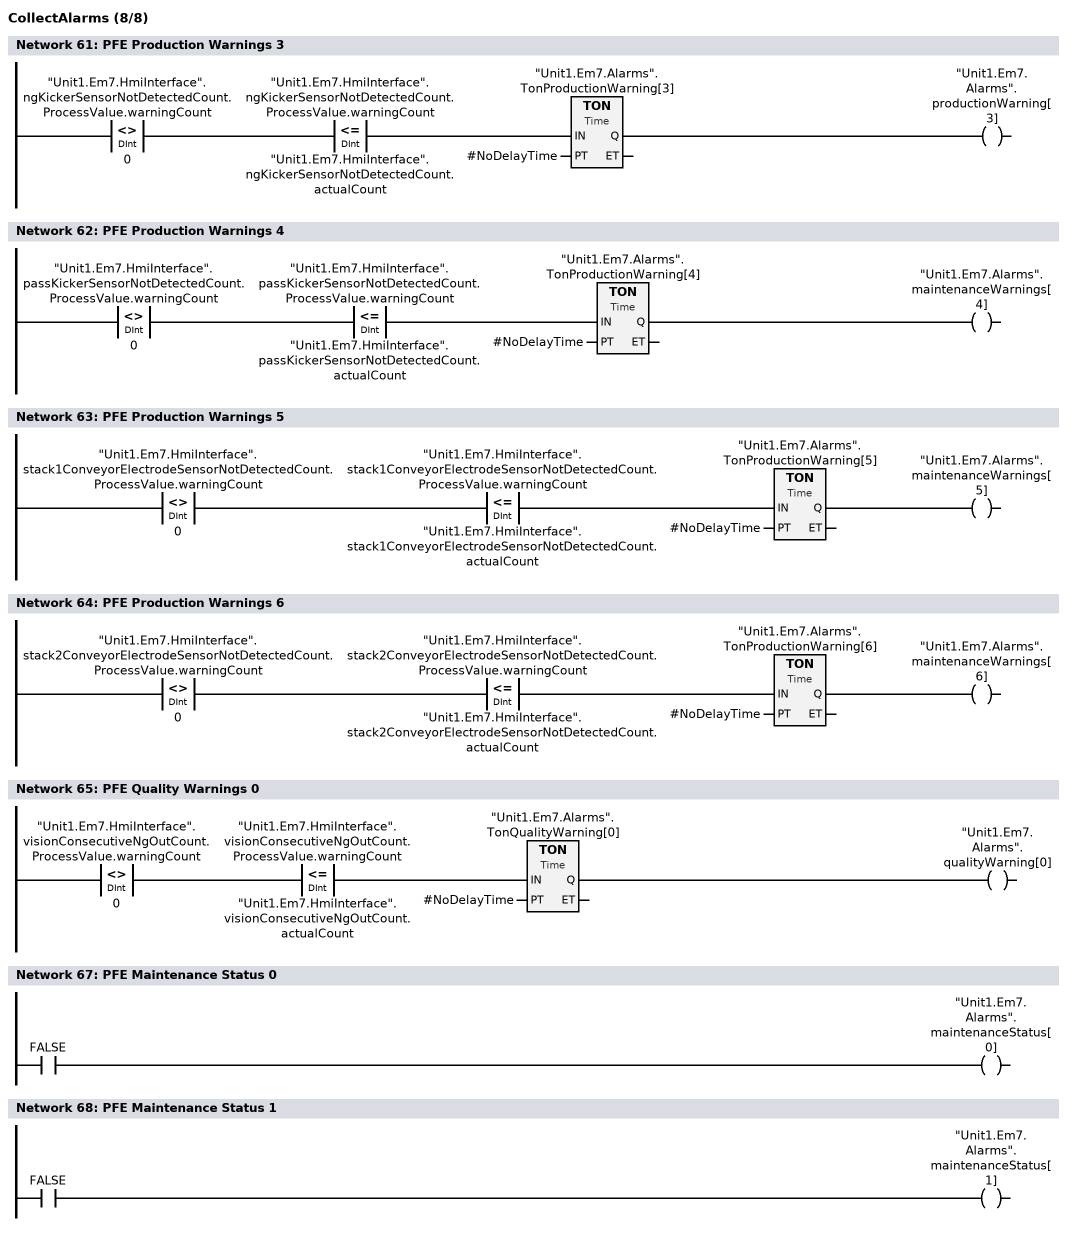
   RUNG wire#powerrail
      { S7_Templates := "SrcType := DInt" } NE_Contact(in1 := "Unit1.Em7.HmiInterface".ngKickerSensorNotDetectedCount.ProcessValue.warningCount, in2 := 0)
      { S7_Templates := "SrcType := DInt" } LE_Contact(in1 := "Unit1.Em7.HmiInterface".ngKickerSensorNotDetectedCount.ProcessValue.warningCount, in2 := "Unit1.Em7.HmiInterface".ngKickerSensorNotDetectedCount.actualCount)
      { S7_Templates := "time_type := Time" } "Unit1.Em7.Alarms".TonProductionWarning[3].TON(pt := #NoDelayTime, et =>)
      Coil( "Unit1.Em7.Alarms".productionWarning[3] )
   END_RUNG
   // the same network as SCL:
   "Unit1.Em7.Alarms".TonProductionWarning[3].TON(IN := ("Unit1.Em7.HmiInterface".ngKickerSensorNotDetectedCount.ProcessValue.warningCount <> 0) AND ("Unit1.Em7.HmiInterface".ngKickerSensorNotDetectedCount.ProcessValue.warningCount <= "Unit1.Em7.HmiInterface".ngKickerSensorNotDetectedCount.actualCount),
                           PT := #NoDelayTime);
   "Unit1.Em7.Alarms".productionWarning[3] := "Unit1.Em7.Alarms".TonProductionWarning[3].Q;
END_REGION

REGION Network 62: PFE Production Warnings 4
   RUNG wire#powerrail
      { S7_Templates := "SrcType := DInt" } NE_Contact(in1 := "Unit1.Em7.HmiInterface".passKickerSensorNotDetectedCount.ProcessValue.warningCount, in2 := 0)
      { S7_Templates := "SrcType := DInt" } LE_Contact(in1 := "Unit1.Em7.HmiInterface".passKickerSensorNotDetectedCount.ProcessValue.warningCount, in2 := "Unit1.Em7.HmiInterface".passKickerSensorNotDetectedCount.actualCount)
      { S7_Templates := "time_type := Time" } "Unit1.Em7.Alarms".TonProductionWarning[4].TON(pt := #NoDelayTime, et =>)
      Coil( "Unit1.Em7.Alarms".maintenanceWarnings[4] )
   END_RUNG
   // the same network as SCL:
   "Unit1.Em7.Alarms".TonProductionWarning[4].TON(IN := ("Unit1.Em7.HmiInterface".passKickerSensorNotDetectedCount.ProcessValue.warningCount <> 0) AND ("Unit1.Em7.HmiInterface".passKickerSensorNotDetectedCount.ProcessValue.warningCount <= "Unit1.Em7.HmiInterface".passKickerSensorNotDetectedCount.actualCount),
                           PT := #NoDelayTime);
   "Unit1.Em7.Alarms".maintenanceWarnings[4] := "Unit1.Em7.Alarms".TonProductionWarning[4].Q;
END_REGION

REGION Network 63: PFE Production Warnings 5
   RUNG wire#powerrail
      { S7_Templates := "SrcType := DInt" } NE_Contact(in1 := "Unit1.Em7.HmiInterface".stack1ConveyorElectrodeSensorNotDetectedCount.ProcessValue.warningCount, in2 := 0)
      { S7_Templates := "SrcType := DInt" } LE_Contact(in1 := "Unit1.Em7.HmiInterface".stack1ConveyorElectrodeSensorNotDetectedCount.ProcessValue.warningCount, in2 := "Unit1.Em7.HmiInterface".stack1ConveyorElectrodeSensorNotDetectedCount.actualCount)
      { S7_Templates := "time_type := Time" } "Unit1.Em7.Alarms".TonProductionWarning[5].TON(pt := #NoDelayTime, et =>)
      Coil( "Unit1.Em7.Alarms".maintenanceWarnings[5] )
   END_RUNG
   // the same network as SCL:
   "Unit1.Em7.Alarms".TonProductionWarning[5].TON(IN := ("Unit1.Em7.HmiInterface".stack1ConveyorElectrodeSensorNotDetectedCount.ProcessValue.warningCount <> 0) AND ("Unit1.Em7.HmiInterface".stack1ConveyorElectrodeSensorNotDetectedCount.ProcessValue.warningCount <= "Unit1.Em7.HmiInterface".stack1ConveyorElectrodeSensorNotDetectedCount.actualCount),
                           PT := #NoDelayTime);
   "Unit1.Em7.Alarms".maintenanceWarnings[5] := "Unit1.Em7.Alarms".TonProductionWarning[5].Q;
END_REGION

REGION Network 64: PFE Production Warnings 6
   RUNG wire#powerrail
      { S7_Templates := "SrcType := DInt" } NE_Contact(in1 := "Unit1.Em7.HmiInterface".stack2ConveyorElectrodeSensorNotDetectedCount.ProcessValue.warningCount, in2 := 0)
      { S7_Templates := "SrcType := DInt" } LE_Contact(in1 := "Unit1.Em7.HmiInterface".stack2ConveyorElectrodeSensorNotDetectedCount.ProcessValue.warningCount, in2 := "Unit1.Em7.HmiInterface".stack2ConveyorElectrodeSensorNotDetectedCount.actualCount)
      { S7_Templates := "time_type := Time" } "Unit1.Em7.Alarms".TonProductionWarning[6].TON(pt := #NoDelayTime, et =>)
      Coil( "Unit1.Em7.Alarms".maintenanceWarnings[6] )
   END_RUNG
   // the same network as SCL:
   "Unit1.Em7.Alarms".TonProductionWarning[6].TON(IN := ("Unit1.Em7.HmiInterface".stack2ConveyorElectrodeSensorNotDetectedCount.ProcessValue.warningCount <> 0) AND ("Unit1.Em7.HmiInterface".stack2ConveyorElectrodeSensorNotDetectedCount.ProcessValue.warningCount <= "Unit1.Em7.HmiInterface".stack2ConveyorElectrodeSensorNotDetectedCount.actualCount),
                           PT := #NoDelayTime);
   "Unit1.Em7.Alarms".maintenanceWarnings[6] := "Unit1.Em7.Alarms".TonProductionWarning[6].Q;
END_REGION

REGION Network 65: PFE Quality Warnings 0
   RUNG wire#powerrail
      { S7_Templates := "SrcType := DInt" } NE_Contact(in1 := "Unit1.Em7.HmiInterface".visionConsecutiveNgOutCount.ProcessValue.warningCount, in2 := 0)
      { S7_Templates := "SrcType := DInt" } LE_Contact(in1 := "Unit1.Em7.HmiInterface".visionConsecutiveNgOutCount.ProcessValue.warningCount, in2 := "Unit1.Em7.HmiInterface".visionConsecutiveNgOutCount.actualCount)
      { S7_Templates := "time_type := Time" } "Unit1.Em7.Alarms".TonQualityWarning[0].TON(pt := #NoDelayTime, et =>)
      Coil( "Unit1.Em7.Alarms".qualityWarning[0] )
   END_RUNG
   // the same network as SCL:
   "Unit1.Em7.Alarms".TonQualityWarning[0].TON(IN := ("Unit1.Em7.HmiInterface".visionConsecutiveNgOutCount.ProcessValue.warningCount <> 0) AND ("Unit1.Em7.HmiInterface".visionConsecutiveNgOutCount.ProcessValue.warningCount <= "Unit1.Em7.HmiInterface".visionConsecutiveNgOutCount.actualCount),
                           PT := #NoDelayTime);
   "Unit1.Em7.Alarms".qualityWarning[0] := "Unit1.Em7.Alarms".TonQualityWarning[0].Q;
END_REGION

REGION Network 66: *************** Status ***************************
END_REGION

REGION Network 67: PFE Maintenance Status 0
   RUNG wire#powerrail
      Contact( FALSE )
      Coil( "Unit1.Em7.Alarms".maintenanceStatus[0] )
   END_RUNG
   // the same network as SCL:
   "Unit1.Em7.Alarms".maintenanceStatus[0] := FALSE;
END_REGION

REGION Network 68: PFE Maintenance Status 1
   RUNG wire#powerrail
      Contact( FALSE )
      Coil( "Unit1.Em7.Alarms".maintenanceStatus[1] )
   END_RUNG
   // the same network as SCL:
   "Unit1.Em7.Alarms".maintenanceStatus[1] := FALSE;
END_REGION
END_FUNCTION
